KUKA KRL data list: style1app1opt1.dat

&ACCESS RVO1
&REL 339
&COMMENT NUT1
&PARAM EDITMASK = *
&PARAM TEMPLATE = C:\KRC\TP\Nutweld\Template\NutWeld_Vorgabe
&PARAM DISKPATH = KRC:\R1\Program\StyleApps\Options
DEFDAT  style1app1opt1
;FOLD EXTERNAL DECLARATIONS;%{PE}%MKUKATPBASIS,%CEXT,%VCOMMON,%P
;FOLD BASISTECH EXT;%{PE}%MKUKATPBASIS,%CEXT,%VEXT,%P
EXT  BAS (BAS_COMMAND  :IN,REAL  :IN )
;ENDFOLD (BASISTECH EXT)
;FOLD NutWeld
;ENDFOLD (NutWeld)
;FOLD USER EXT;%{E}%MKUKATPUSER,%CEXT,%VEXT,%P
;Make here your modifications
;ENDFOLD (USER EXT)
DECL E6POS XP20={X -3850.82104,Y -108.397034,Z -435.544800,A -178.432037,B 0.654220462,C -179.967712,S 2,T 34,E1 0.0,E2 0.0,E3 0.0,E4 0.0,E5 0.0,E6 0.0}
DECL FDAT FP20={TOOL_NO 1,BASE_NO 3,IPO_FRAME #BASE,POINT2[] " ",TQ_STATE FALSE}
;ENDFOLD (EXTERNAL DECLARATIONS)








DECL FDAT FPNW1={TOOL_NO 2,BASE_NO 1,IPO_FRAME #TCP,POINT2[] " ",TQ_STATE FALSE}
DECL E6POS XPNW1={X 123.774101,Y 312.995331,Z -88.6478,A 8.71582699,B 8.82717705,C 1.11576855,S 2,T 3,E1 0.0,E2 0.0,E3 0.0,E4 0.0,E5 0.0,E6 0.0}
DECL NutWeld_SUGG_T LAST_NutWeld={POINT1[] "PNW1_SPOT7              ",POINT2[] "PNW0                    ",CP_PARAMS[] "CPDATNutWeld0           ",PTP_PARAMS[] "PDATNutWeld0            ",CONT[] "C_PTP                   ",CP_VEL[] "2                       ",PTP_VEL[] "100                     ",SYNC_PARAMS[] "SYNCDAT                 ",SPL_NAME[] "S0                      ",NutWeld_PARAMS[] "NutData1_7              ",GunNr 1,SpotNr 7,Offset 45}
DECL BASIS_SUGG_T LAST_BASIS={POINT1[] "P0                      ",POINT2[] "P0                      ",CP_PARAMS[] "CPDAT0                  ",PTP_PARAMS[] "PDAT0                   ",CONT[] "                        ",CP_VEL[] "2                       ",PTP_VEL[] " 100                    ",SYNC_PARAMS[] "SYNCDAT                 ",SPL_NAME[] "S0                      ",A_PARAMS[] "ADAT0                   "}
DECL PDAT PPDAT0={VEL 100.000,ACC 100.000,APO_DIST 100.000,APO_MODE #CDIS,GEAR_JERK 50.0000,EXAX_IGN 0}
DECL E6POS XP0={X -3704.29346,Y 1.10223198,Z -449.805786,A -178.368118,B 0.266879767,C 179.968445,S 2,T 34,E1 0.0,E2 0.0,E3 0.0,E4 0.0,E5 0.0,E6 0.0}
DECL FDAT FP0={TOOL_NO 1,BASE_NO 3,IPO_FRAME #TCP,POINT2[] " ",TQ_STATE FALSE}
DECL MODULEPARAM_T LAST_TP_PARAMS={PARAMS[] "NutWeld_CmdPos=Weld; NutWeld_Move=LIN; NutWeld_NutWeldDat=NutData1_7; NutWeld_NWGunNr=1; NutWeld_NWSpotNr=7; NutWeld_NWOffset=45; Kuka.MoveDataName=gAboveWeld; Kuka.VelocityPath=2; Kuka.PointName=PNW1_CNTRH_SPOT7; Kuka.BlendingEnabled=False; Kuka.FrameData.tq_state=False; Kuka.FrameData.base_no=1; Kuka.FrameData.tool_no=1; Kuka.FrameData.ipo_frame=#TCP; Kuka.FrameData.point2=; Kuka.MovementData.apo_fac=50; Kuka.MovementData.apo_dist=100; Kuka.MovementData.axis_acc=100; Kuka.MovementData.axis_vel=100; Kuka.MovementData.circ_typ=#BASE; Kuka.MovementData.exax_ign=0; Kuka.MovementData.jerk_fac=50; Kuka.MovementData.ori_typ=#VAR; Kuka.MovementData.acc=100; Kuka.MovementData.gear_jerk=50  "}
DECL E6POS XP8={X -3704.29346,Y 1.10223198,Z -449.805786,A -178.368118,B 0.266879767,C 179.968445,S 2,T 34,E1 0.0,E2 0.0,E3 0.0,E4 0.0,E5 0.0,E6 0.0}
DECL FDAT FP8={TOOL_NO 1,BASE_NO 3,IPO_FRAME #TCP,POINT2[] " ",TQ_STATE FALSE}
DECL LDAT LCPDAT8={VEL 2.00000,ACC 100.000,APO_DIST 100.000,APO_FAC 50.0000,AXIS_VEL 100.000,AXIS_ACC 100.000,ORI_TYP #VAR,CIRC_TYP #BASE,JERK_FAC 50.0000,GEAR_JERK 50.0000,EXAX_IGN 0}
DECL LDAT LCPDAT12={VEL 2.00000,ACC 100.000,APO_DIST 100.000,APO_FAC 50.0000,AXIS_VEL 100.000,AXIS_ACC 100.000,ORI_TYP #VAR,CIRC_TYP #BASE,JERK_FAC 50.0000,GEAR_JERK 50.0000,EXAX_IGN 0}
DECL LDAT LCPDAT16={VEL 2.00000,ACC 100.000,APO_DIST 100.000,APO_FAC 50.0000,AXIS_VEL 100.000,AXIS_ACC 100.000,ORI_TYP #VAR,CIRC_TYP #BASE,JERK_FAC 50.0000,GEAR_JERK 50.0000,EXAX_IGN 0}
DECL LDAT LCPDAT17={VEL 2.00000,ACC 100.000,APO_DIST 100.000,APO_FAC 50.0000,AXIS_VEL 100.000,AXIS_ACC 100.000,ORI_TYP #VAR,CIRC_TYP #BASE,JERK_FAC 50.0000,GEAR_JERK 50.0000,EXAX_IGN 0}
DECL PDAT PPDAT18={VEL 100.000,ACC 100.000,APO_DIST 100.000,APO_MODE #CDIS,GEAR_JERK 50.0000,EXAX_IGN 0}
DECL E6POS XP19={X -3851.81445,Y -107.010963,Z -442.857483,A -178.432037,B 0.654220223,C -179.967712,S 2,T 34,E1 0.0,E2 0.0,E3 0.0,E4 0.0,E5 0.0,E6 0.0}
DECL FDAT FP19={TOOL_NO 1,BASE_NO 3,IPO_FRAME #BASE,POINT2[] " ",TQ_STATE FALSE}
DECL LDAT LCPDAT18={VEL 2.00000,ACC 100.000,APO_DIST 100.000,APO_FAC 50.0000,AXIS_VEL 100.000,AXIS_ACC 100.000,ORI_TYP #VAR,CIRC_TYP #BASE,JERK_FAC 50.0000,GEAR_JERK 50.0000,EXAX_IGN 0}
ENDDAT
